INTERFACE I_MotionPowerTask EXTENDS I_MotionTask, I_AxisEnable

END_INTERFACE

(* stored: Version 1.1.0.1, ProductVersion 3.1.4026.18
   Itf I_MotionPowerTask: Id {e184382f-6a50-4582-a666-471c66e3455d} *)
